// TIA Portal V18 export
DATA_BLOCK "ChaosDB"   // DB18
{ S7_Optimized_Access := 'TRUE' }
VERSION : 0.1
// stored: AutoNumber true, DBAccessibleFromOPCUA true, IsOnlyStoredInLoadMemory false, IsRetainMemResEnabled false, IsWriteProtectedInAS false, MemoryReserve 100
   VAR
      Step0 { ExternalAccessible := 'False'; ExternalVisible := 'False'; ExternalWritable := 'False'} : Bool;
      Step1 { ExternalAccessible := 'False'; ExternalVisible := 'False'; ExternalWritable := 'False'} : Bool;
      Step2 { ExternalAccessible := 'False'; ExternalVisible := 'False'; ExternalWritable := 'False'} : Bool;
      Step3 { ExternalAccessible := 'False'; ExternalVisible := 'False'; ExternalWritable := 'False'} : Bool;
      Step4 : Bool;
      Step5 : Bool;
      Step6 : Bool;
      Step7 : Bool;
      Step10 : Bool;
      Step20 : Bool;
      Step21 : Bool;
      Step1_Step2 { ExternalAccessible := 'False'; ExternalVisible := 'False'; ExternalWritable := 'False'} : Bool;
      Step2_Step3 { ExternalAccessible := 'False'; ExternalVisible := 'False'; ExternalWritable := 'False'} : Bool;
      Step2_Step5 : Bool;
      Step4_Step5 : Bool;
      Step2_Step20 : Bool;
      Step3_Step_4 : Bool;
      Step4_Step6 : Bool;
      Step4_Step10 : Bool;
      Step4_Step20 : Bool;
      Step5_Step2 : Bool;
      Step6_Step7 : Bool;
      Step7_Step4 : Bool;
      Step10_Step2 : Bool;
      Step20_Step21 : Bool;
      Step21_Step2 : Bool;
      Edge_Step1M { ExternalAccessible := 'False'; ExternalVisible := 'False'; ExternalWritable := 'False'} : Bool;
      Edge_Step1S : Bool;
      Edge_Reset_Z2_M : Bool;
      Edge_Reset_Z2_S : Bool;
      Edge_Reset_X_S : Bool;
      Edge_Reset_X_M : Bool;
      Edge_Reset_Y_S : Bool;
      Edge_Reset_Y_M : Bool;
      Reset_error_main : Bool;
      Edge_M_res_err_main : Bool;
      Edge_S_res_err_main : Bool;
      Edge_Reset_Z1_S : Bool;
      Edge_Reset_Z1_M : Bool;
      Monitor_state : Bool;   // Auxiliary variable
      Edge_S_ResCMMOZ2 : Bool;   // Reset CMMO Z2 Controller
      Edge_M_ResCMMOZ2 : Bool;   // Reset CMMO Z2 Controller
      Restart_CMMO_Z2_Cmd : Bool;   // Reset CMMO Z2 Controller
      Edge_S_ResCMMOZ1 : Bool;   // Reset CMMO Z1Controller
      Edge_M_ResCMMOZ1 : Bool;   // Reset CMMO Z1 Controller
      Restart_CMMO_Z1_Cmd : Bool;   // Reset CMMO Z1Controller
      Edge_S_ResCMMPX : Bool;   // Reset CMMP X Controller
      Edge_M_ResCMMPX : Bool;   // Reset CMMP X Controller
      Restart_CMMP_X_Cmd : Bool;   // Reset CMMP X Controller
      Edge_S_ResCMMPY : Bool;   // Reset CMMP Y Controller
      Edge_M_ResCMMPY : Bool;   // Reset CMMP Y Controller
      Restart_CMMP_Y_Cmd : Bool;   // Reset CMMP Y Controller
      Z2_Stop_E : Bool;
      Z2_Stop_EM : Bool;
   END_VAR
BEGIN
END_DATA_BLOCK
